Fanuc TP program (LS listing): 04_camera_minute_wait.ls

/PROG MOVE_HOME_CAMERA_INSPECT
/ATTR
OWNER = MNEDITOR;
COMMENT = "auto";
/MN
   1:  UFRAME_NUM=1 ;
   2:  UTOOL_NUM=1 ;
   3:  !Move from home to camera inspection pose, enable camera, wait 60s, disable camera, return home ;
   4:  J PR[1:home] 100% FINE ;
   5:  L PR[17:camera inspection pose] 100mm/sec CNT50 ;
   6:  DO[1:camera on]=ON ;
   7:  WAIT 60.00(sec) ;
   8:  DO[1]=OFF ;
   9:  J PR[1:home] 100% FINE ;
/POS
/END
